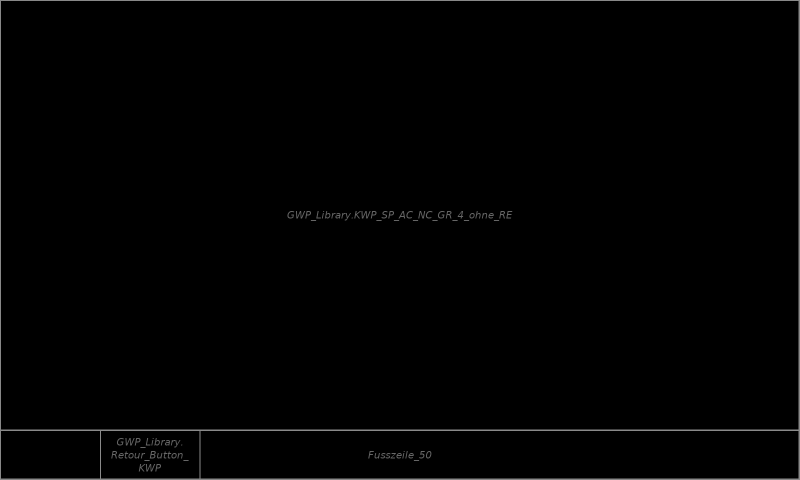
VISUALIZATION KWP_SP_AC_NC_GR_4_ohne_RE  // 800x480
    Frame (0,0 800x430)
        shows GWP_Library.KWP_SP_AC_NC_GR_4_ohne_RE(FB_GR_4_ohne_RE := Main.KWP_SP_AC_NC_0.GR_4_ohne_RE_0)
    Group (0,430 800x50)
        Frame (0,0 800x50)
            shows Fusszeile_50()
        Frame (100,0 100x50)
            shows GWP_Library.Retour_Button_KWP()
END_VISUALIZATION

(* stored: Version 1.1.0.1, ProductVersion 3.1.4022.6
   Visu KWP_SP_AC_NC_GR_4_ohne_RE: Id {a48cee1b-9fe8-4917-a5c2-2405e8c47063} *)
